(* CODESYS project 05_MySQL_DB_External.ecp

Project tree, tasks and I/O mapping:
  PFC_MySQL_DB_External : 750-8212 PFC200 G2 2ETH RS, WAGO, order no. 0750-8212, version 5.16.3.16
    application Application
      libraries: WagoAppTime, 1.7.3.3 (WAGO); VisuDialogs, * (System); WagoAppSQL_MySQL, 1.6.1.0 (WAGO)
      task PLC_Task (cyclic, interval t#30ms, priority 13) calls PLC_PRG
      task Task_SQL (cyclic, interval t#10ms, priority 14) calls PRG_SQL
      task VISU_TASK (cyclic, interval 100 ms, priority 15) calls VisuElems.Visu_Prg
      program PLC_PRG [ST]
      program PRG_SQL [FBD]: actScanner
      FBs/
        function block FbSQLInsertCommand_dbTraining_Format9 [ST]
      visualisation Database
      visualisation phpMyAdmin
      data type typByte2String
      visualisation visuQueryResult
      data type typState
    ProjectConfiguration
    ProjectConfigurationTxt
    Kbus : Kbus, WAGO, version 1.4.0.2
        unmapped channels: K-BUS diagnostics
    MODBUS
      MODBUS : MODBUS, WAGO, order no. n/a, version 1.1.1.16
    Serial
      COM1 : COM1, WAGO, version 0.0.0.19
    Common.PCI
    EtherNet/IP
      Ethernet : Ethernet, WAGO, version 35.16.0.0
  libraries: VisuSymbols, 3.5.10.0 (System); WagoVisuIcons, 1.1.0.3 (WAGO)
  text list GlobalTextList
  00000000-0000-0000-0000-000000000000|C:\Users\MarkusF\AppData\Local\Temp\47851c6884b74d138d157e768835671a\Project.xml
  00000000-0000-0000-0000-000000000000|C:\Users\MarkusF\AppData\Local\Temp\be8271bb544c4b49a55d0a08df03c384\ProjectCfg.txt
*)

// PFC_MySQL_DB_External/Application/typByte2String
TYPE typByte2String :
UNION		// convert an array of byte to a readable string
	sData:	STRING(MYSQL_MAX_ROW_SIZE);
	abData:	ARRAY [0..MYSQL_MAX_ROW_SIZE] OF BYTE;
END_UNION
END_TYPE

// PFC_MySQL_DB_External/Application/typState
{attribute 'qualified_only'}
{attribute 'strict'}
TYPE typState :
(
	eIdle,
	eHandleLogin,
	eProcessSqlExecute,
	eHandleLogout,
	eErrorHandling
);
END_TYPE

// PFC_MySQL_DB_External/Application/PLC_PRG
PROGRAM PLC_PRG
VAR
	timDelay			: TON;
	dtLocalTime			: DATE_AND_TIME;
	sTime				: STRING(8);
	sDate				: STRING(10);

	xRandomActive		: BOOL := TRUE;
	rOffsetTemperature	: REAL;
	rOffsetVoltage		: REAL;
	xDigitalInput8		: BOOL;

	rTemperatureStatic	: REAL := 23.5;
	rVoltageStatic		: REAL := 5.834;
	rTemperature		: REAL;
	rVoltage			: REAL;
END_VAR

// get date and time of the controller only every second, because it's stressy
timDelay(IN := NOT timDelay.Q, PT := T#1S);
IF timDelay.Q THEN
	dtLocalTime	:= FuGetLocalDateAndTime();
	sTime		:= WagoAppString.FuTodToString(bFormat := 1, todInput := TO_TOD(dtLocalTime));
	sDate		:= WagoAppString.FuDateToString(bFormat := 0, datInput := TO_DATE(dtLocalTime));

	// generate some data to fill database
	IF xRandomActive THEN
		// create some randomness for temperature value
		rOffsetTemperature	:= 8.34 * SIN(TO_REAL(PRG_SQL.a) / 30.0);
		// create some randomness for voltage value
		rOffsetVoltage		:= 3.78 * SIN(TO_REAL(PRG_SQL.a) / 12.8);
	ELSE
		rOffsetVoltage		:= 0;
		rOffsetTemperature	:= 0;
	END_IF
	
	// toggle input
	xDigitalInput8			:= NOT xDigitalInput8;
END_IF;

// add some changes
rTemperature	:= rTemperatureStatic 	+ rOffsetTemperature;
rVoltage		:= rVoltageStatic		+ rOffsetVoltage;

END_PROGRAM

// PFC_MySQL_DB_External/Application/PRG_SQL
PROGRAM PRG_SQL
VAR
//	program is alive
	a					: UDINT;

//	MySQL Database called ___"dbTraining"___
//	with phpMyAdmin on Linux-PC
//	Tablename: ___________"TblTrainingData"__________

	sIP_LinuxDB			: STRING := '192.168.1.123';
	sUserLinuxDB		: STRING := 'dozent';
	sPwdLinuxDB			: STRING := 'Master!';
	sDatabaseName		: STRING := 'dbTraining';
	sTableName			: STRING := 'TblTrainingData';

//_______________________________________________________________

	oFBdbTraining_Format9: FbSQLInsertCommand_dbTraining_Format9;
	xConnect			: BOOL;
	sDate				: STRING := 'Date';
	sTime				: STRING := 'Time';
	sTemp				: STRING := 'Temperature';
	sDigitalInput		: STRING := 'EmergencyStop';
	sVoltage			: STRING := 'Voltage';
	xTriggerWrite		: BOOL;
	xConnectedToLinuxDatabase: BOOL;

	FbMySqlQuery		: FbMySql_Query;
	aSqlCommand			: ARRAY [0..MYSQL_SQL_UPPER_BOUND] OF STRING(MYSQL_SQL_LENGTH)
						:= ['SELECT * FROM dbTraining.TblTrainingData WHERE EmergencyStop =  1 AND Date > $272020-01-20$27 LIMIT 10', 10('')];
	xTriggerQuery		: BOOL;
	typResultSqlQuery	: typMySql_ResultSet;
	xBusyQuery			: BOOL;
	xErrorQuery			: BOOL;
	oStatusQuery		: WagoSysErrorBase.FbResult;
	sStatusQuery		: STRING(200);

	iRowQuery			: INT := 3;
	iColQuery			: INT := 3;
	sValueQuery			: STRING(500);
	dwQuery				: DWORD;
	
	uByte2String		: typByte2String;
	
	// scanner
	iRowScanner1,
	iRowScanner2,
	iColScanner			: INT;
	asValueScanner		: ARRAY[1..6, 1..20] OF STRING(500);
	dwQueryScanner		: DWORD;
END_VAR

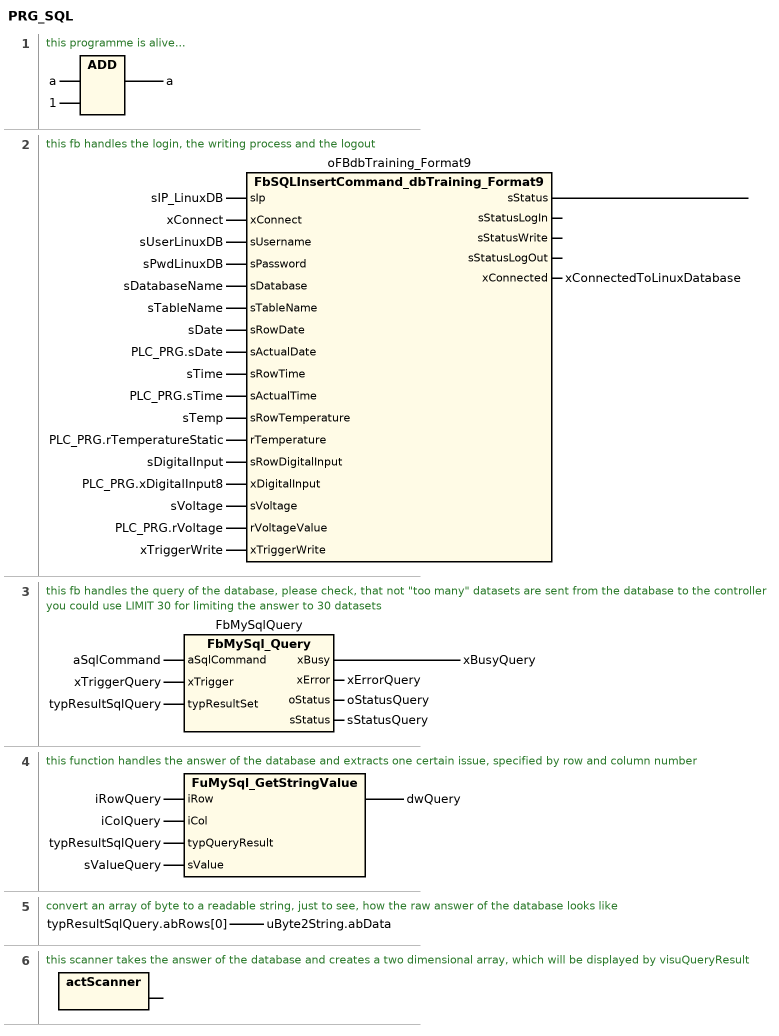
// NETWORK 1
// this programme is alive...
a := a + 1;

// NETWORK 2
// this fb handles the login, the writing process and the logout
oFBdbTraining_Format9(
    sIp := sIP_LinuxDB,
    xConnect := xConnect,
    sUsername := sUserLinuxDB,
    sPassword := sPwdLinuxDB,
    sDatabase := sDatabaseName,
    sTableName := sTableName,
    sRowDate := sDate,
    sActualDate := PLC_PRG.sDate,
    sRowTime := sTime,
    sActualTime := PLC_PRG.sTime,
    sRowTemperature := sTemp,
    rTemperature := PLC_PRG.rTemperatureStatic,
    sRowDigitalInput := sDigitalInput,
    xDigitalInput := PLC_PRG.xDigitalInput8,
    sVoltage := sVoltage,
    rVoltageValue := PLC_PRG.rVoltage,
    xTriggerWrite := xTriggerWrite,
    xConnected => xConnectedToLinuxDatabase); // FbSQLInsertCommand_dbTraining_Format9

// NETWORK 3
// this fb handles the query of the database, please check, that not "too many" datasets are sent from the database to the controller
// you could use LIMIT 30 for limiting the answer to 30 datasets
FbMySqlQuery(
    aSqlCommand := aSqlCommand,
    xTrigger := xTriggerQuery,
    typResultSet := typResultSqlQuery,
    xError => xErrorQuery,
    oStatus => oStatusQuery,
    sStatus => sStatusQuery); // FbMySql_Query
xBusyQuery := FbMySqlQuery.xBusy;

// NETWORK 4
// this function handles the answer of the database and extracts one certain issue, specified by row and column number
dwQuery := FuMySql_GetStringValue(iRow := iRowQuery, iCol := iColQuery, typQueryResult := typResultSqlQuery, sValue := sValueQuery);

// NETWORK 5
// convert an array of byte to a readable string, just to see, how the raw answer of the database looks like
uByte2String.abData := typResultSqlQuery.abRows[0];

// NETWORK 6
// this scanner takes the answer of the database and creates a two dimensional array, which will be displayed by visuQueryResult
actScanner();

ACTION actScanner:
IF dwQuery = 0 THEN
	FOR iRowScanner1 := 1 TO 20 DO
		FOR iColScanner := 1 TO 6 DO
			dwQueryScanner := FuMySql_GetStringValue(
				iRow			:= iRowScanner1,
				iCol			:= iColScanner,
				typQueryResult	:= typResultSqlQuery,
				sValue			:= asValueScanner[iColScanner, iRowScanner1]);
			IF dwQueryScanner <> 0 THEN
				// delete rest of the table
				FOR iRowScanner2 := iRowScanner1 TO 20 DO
					FOR iColScanner := 1 TO 6 DO
						asValueScanner[iColScanner, iRowScanner2] := '';
					END_FOR
				END_FOR
				RETURN;
			END_IF
		END_FOR
	END_FOR
END_IF
END_ACTION

END_PROGRAM

// PFC_MySQL_DB_External/Application/FBs/FbSQLInsertCommand_dbTraining_Format9
FUNCTION_BLOCK FbSQLInsertCommand_dbTraining_Format9
VAR_INPUT
	sIp					: STRING := '192.168.1.2';				// ip address of the server
	xConnect			: BOOL;					// connect to the data base
	sUsername			: STRING;				// database username
	sPassword			: STRING;				// database password
	sDatabase			: STRING;				// database name which you want to acccess
	sTableName			: STRING;				// table which belongs to your chosen database 
	
	sRowDate			: STRING;				// first row of your table
	sActualDate			: STRING(10);
	
	sRowTime			: STRING;				// second row of your table
	sActualTime			: STRING(8);
	
	sRowTemperature		: STRING;				// third row of your table
	rTemperature		: REAL;
	
	sRowDigitalInput	: STRING;				// fourth row of your table
	xDigitalInput		: BOOL;
	
	sVoltage			: STRING;				// fifth row of your table
	rVoltageValue		: REAL;
END_VAR
VAR_OUTPUT
	sStatus				: STRING;
	sStatusLogIn		: STRING(200);
	sStatusWrite		: STRING(200);
	sStatusLogOut		: STRING(200);
	xConnected			: BOOL;
END_VAR
VAR_IN_OUT
	xTriggerWrite		: BOOL;
END_VAR
VAR
	xInit				: BOOL := TRUE;
	aSqlCommand			: ARRAY [0..MYSQL_SQL_UPPER_BOUND] OF STRING(MYSQL_SQL_LENGTH);
	sActualDigitalInput	: STRING(20);

	iState				: INT;
	fbSqlLogin01		: FbMySql_Login;
	xTriggerLogin		: BOOL;
	xBusyLogIn			: BOOL;
	xErrorLogIn			: BOOL;
	
	fbSqlExecute01		: FbMySql_Execute;
	
	xBusyWrite			: BOOL;
	xErrorWrite			: BOOL;
	
	fbSqlLogout01		: FbMySql_Logout;
	xTriggerLogout		: BOOL;
	xBusyLogOut			: BOOL;
	xErrorLogOut		: BOOL;
END_VAR

// initialisation procedure
IF xInit THEN
	aSqlCommand[0] := Format6(
		sFormat	:= 'INSERT INTO %s(%s,%s,%s,%s,%s) ',
		p1		:= ADR(sTableName),
		p2		:= ADR(sRowDate),
		p3		:= ADR(sRowTime),
		p4		:= ADR(sRowTemperature),
		p5		:= ADR(sRowDigitalInput),
		p6		:= ADR(sVoltage));
	xInit := FALSE;			// initialisation process is over
END_IF

//---------------------------------------------------------------------------------------------------------------------------------------------------------------------------------------------------------------------------------------
// since Format5 uses pointers it is necessary to use variables after typecasting- otherwise an error will occur
sActualDigitalInput	:= TO_STRING(xDigitalInput);

aSqlCommand[1] := Format5(
	sFormat	:= 'VALUES($27%s$27,$27%s$27,%4.1f,%s,%5.2f)',		// $27 ==> ' ==> inverted comma
	p1		:= ADR(sActualDate),
	p2		:= ADR(sActualTime),
	p3		:= ADR(rTemperature),
	p4		:= ADR(sActualDigitalInput),
	p5		:= ADR(rVoltageValue));

// target: INSERT INTO 'dbTraining'('Date','Time','Temperature',EmergencyStop,'Voltage') VALUES('2017-10-31',10:33:05,23.3,true,8.7)

// ATTENTION: The function block Login01 has to be called within every PLC cycle!!!
fbSqlLogin01(
	sHost		:= sIp,
	//uiPort	:= ,
	sUsername	:= sUsername,
	sPassword	:= sPassword,
	sDatabase	:= sDatabase,
	xTrigger	:= xTriggerLogin,
	xBusy		=> xBusyLogIn,
	xError		=> xErrorLogIn,
	//oStatus	=> ,
	sStatus		=> sStatusLogIn,
	xConnected	=> xConnected);

CASE iState OF
//------------------------------------------------------------------------------------------
	typState.eIdle:
		sStatus := 'SQL idle';
		IF xConnect THEN
			xTriggerLogin := TRUE;
			iState := typState.eHandleLogin;
		END_IF

//------------------------------------------------------------------------------------------
	typState.eHandleLogin:
		IF NOT xTriggerLogin THEN
			IF xConnected THEN
				iState	:= typState.eProcessSqlExecute;
				sStatus	:= 'SQL connected';
			ELSE
				iState	:= typState.eErrorHandling;
				sStatus	:= 'SQL connect error';
			END_IF
		END_IF
//------------------------------------------------------------------------------------------	
	typState.eProcessSqlExecute:
		fbSqlExecute01(
			aSqlCommand	:= aSqlCommand,
			xTrigger	:= xTriggerWrite,
			xBusy		=> xBusyWrite,
			xError		=> xErrorWrite,
			//oStatus	=> ,
			sStatus		=> sStatusWrite);
		IF NOT xConnect THEN
			xTriggerLogout := TRUE;
			iState := typState.eHandleLogout;
		END_IF

//------------------------------------------------------------------------------------------	
	typState.eHandleLogout:
		fbSqlLogout01(
			xTrigger	:= xTriggerLogout,
			xBusy		=> xBusyLogOut,
			xError		=> xErrorLogOut,
			//oStatus	=> ,
			sStatus		=> sStatusLogOut);
		IF NOT xTriggerLogout THEN
			IF NOT xErrorLogOut THEN
				iState	:= typState.eIdle;
				sStatus	:= 'SQL disconnected';
			ELSE
				iState	:= typState.eErrorHandling;
				sStatus	:= 'SQL Logout Error';
			END_IF;
		END_IF;
	typState.eErrorHandling:
		sStatus := 'Error Handling!!!';

END_CASE
//------------------------------------------------------------------------------------------

END_FUNCTION_BLOCK

// PFC_MySQL_DB_External/Application/Database
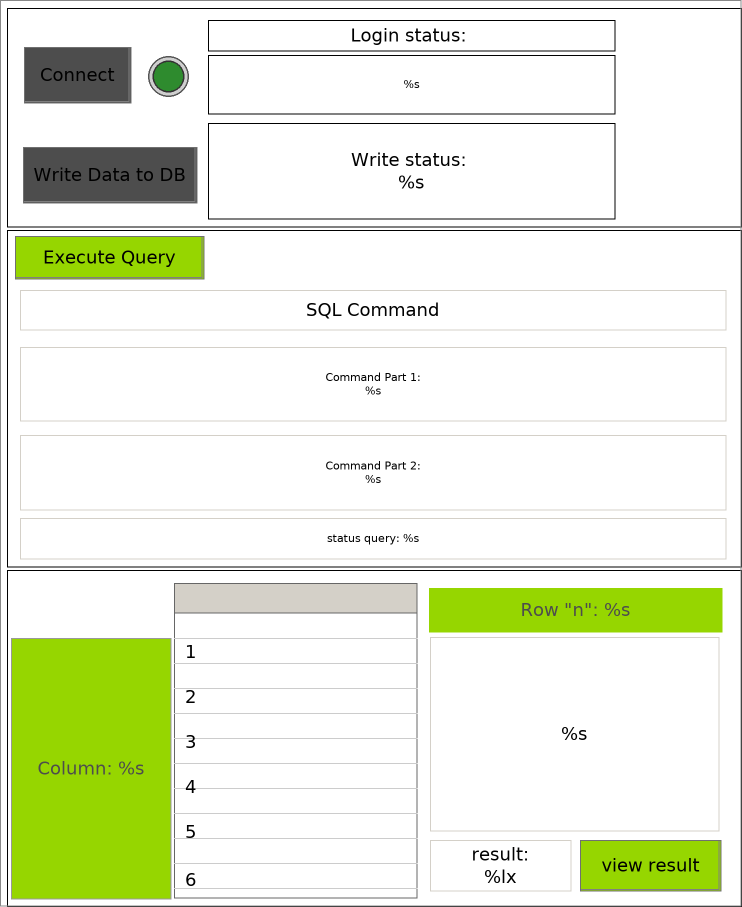
VISUALIZATION Database  // 742x907
    Rectangle (7,230 735x337)
    Button (15,236 189x43), "Execute Query", input disabled if: NOT PRG_SQL.oFBdbTraining_Format9.xConnected
        tap PRG_SQL.xTriggerQuery
    Textfield (20,347 706x74), "Command Part 1: %s", text variable: PRG_SQL.aSqlCommand[0]
        OnMouseClick: write the text variable via Edit
    Textfield (20,435 706x75), "Command Part 2: %s", text variable: PRG_SQL.aSqlCommand[1]
        OnMouseClick: write the text variable via Edit
    Rectangle (7,8 735x219)
    Button (24,47 107x56), "Connect"
        toggle PRG_SQL.xConnect
    Lamp1 (145,52 47x49), variable: PRG_SQL.oFBdbTraining_Format9.xConnected, style: Lamp-Lamp1-Green
    Group (208,20 516x199)
        Rectangle (0,103 407x96), "Write status: %s", text variable: PRG_SQL.oFBdbTraining_Format9.sStatusWrite
        Rectangle (0,0 407x31), "Login status:"
        Rectangle (0,35 407x59), "%s", text variable: PRG_SQL.oFBdbTraining_Format9.sStatusLogIn
    Button (23,147 174x56), "Write Data to DB", input disabled if: NOT PRG_SQL.oFBdbTraining_Format9.xConnected
        toggle PRG_SQL.xTriggerWrite
    Rectangle (7,570 735x337)
    Rectangle (429,588 293x44), "Row "n": %s", tooltip "Row max depends on your query default: 100", text variable: PRG_SQL.iRowQuery
        OnMouseClick: write the text variable via Edit, min 1, max 100
    Rectangle (11,638 160x261), "Column: %s", tooltip "Column max = 6", text variable: PRG_SQL.iColQuery
        OnMouseClick: write the text variable via Edit, min 0, max 6
    Textfield (430,637 289x194), "%s", text variable: PRG_SQL.sValueQuery
    Table (174,583 243x315), data array: PRG_SQL.typResultSqlQuery.astColumns
        p3854506369: PRG_SQL.typResultSqlQuery.astColumns[INDEX].sName
        p1892666644: PRG_SQL.typResultSqlQuery.astColumns[INDEX].udiLength
        p338671338: PRG_SQL.typResultSqlQuery.astColumns[INDEX].eType
        p2170511999: PRG_SQL.typResultSqlQuery.astColumns[INDEX].wFlags
        p3723444502: PRG_SQL.typResultSqlQuery.astColumns[INDEX].bDecimals
        p2232123230: dbTraining Data
    Rectangle (173,630 36x44), "1"
    Rectangle (173,675 36x44), "2"
    Rectangle (173,720 36x44), "3"
    Rectangle (173,765 36x44), "4"
    Rectangle (173,810 36x44), "5"
    Rectangle (173,858 36x44), "6"
    Textfield (20,518 706x41), "status query: %s", text variable: PRG_SQL.sStatusQuery
    Textfield (20,290 706x40), "SQL Command"
    Textfield (430,840 141x51), "result: %lx", text variable: PRG_SQL.dwQuery
    Button (580,840 141x51), "view result", input disabled if: PRG_SQL.dwQuery <> 0
        OnMouseClick:  Assign=visuQueryResult, Type=Assignment
END_VISUALIZATION

// PFC_MySQL_DB_External/Application/phpMyAdmin
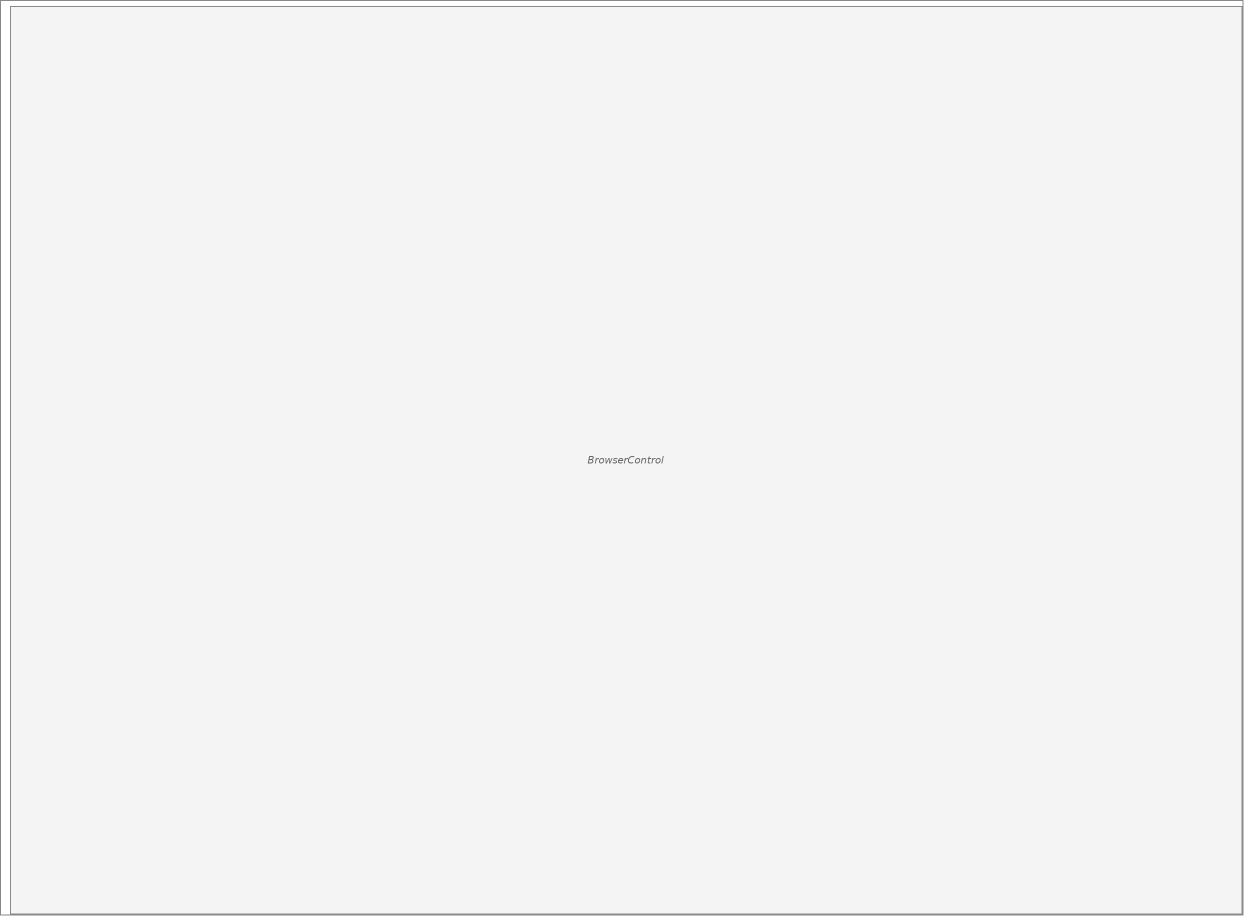
VISUALIZATION phpMyAdmin  // 1244x916
    BrowserControl (10,6 1232x908)
        p3734058945: 'http://192.168.1.1/phpMyAdmin/index.php'
END_VISUALIZATION

// PFC_MySQL_DB_External/Application/visuQueryResult
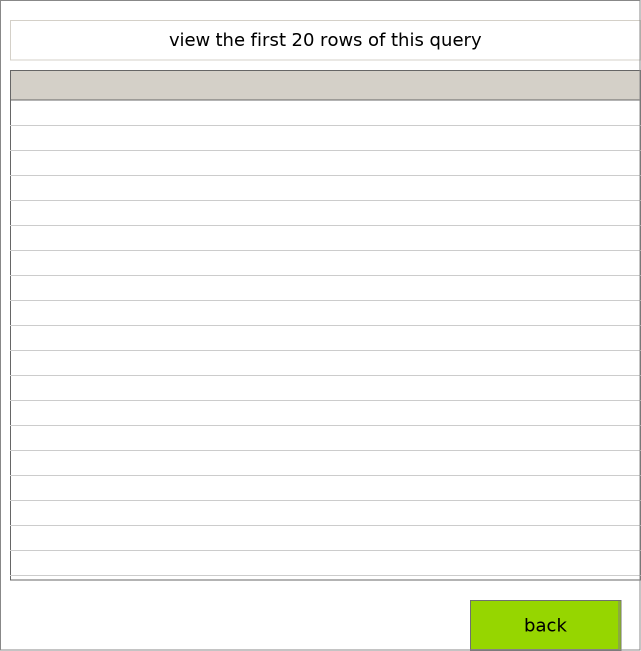
VISUALIZATION visuQueryResult  // 641x651
    Table (10,70 631x510), data array: PRG_SQL.asValueScanner
        p3854506369: PRG_SQL.asValueScanner[1,INDEX]
        p1892666644: PRG_SQL.asValueScanner[2,INDEX]
        p338671338: PRG_SQL.asValueScanner[3,INDEX]
        p2170511999: PRG_SQL.asValueScanner[4,INDEX]
        p3723444502: PRG_SQL.asValueScanner[5,INDEX]
        p1218418051: PRG_SQL.asValueScanner[6,INDEX]
        p2232123230: No.
        p511219082: Date
        p1755163831: Time
        p4092479075: Temp.
        p2237128397: E-Stop
        p505689113: Voltage
    Button (470,600 151x51), "back"
        OnMouseClick:  Assign=Database, Type=Assignment
    Textfield (10,20 631x40), "view the first 20 rows of this query"
END_VISUALIZATION
